Fanuc KAREL source: kt00308.KL

PROGRAM KT00308
%STACKSIZE=65535
%PRIORITY=65535
%NOLOCKGROUP
VAR
H1 : ARRAY[2] OF SHORT
R2 : REAL
OUT : BOOLEAN
BEGIN
H1[1]=2
R2=3.0
OUT=(R2 <> (H1[1]))
END KT00308
